// TIA Portal V20 export
TYPE "LBP_typeModularMcpUniversalInput"
TITLE = Modular MCP image / Image MCP modulaire
// Input image of universal keypad for modular MCP / Image des entrées du pupitre universel pour MCP modulaires
   STRUCT
      key0 : Bool;   // input image n+0 bit 0 / Image des entrées n+0 bit 0
      key1 : Bool;   // input image n+0 bit 1 / Image des entrées n+0 bit 1
      key2 : Bool;   // input image n+0 bit 2 / Image des entrées n+0 bit 2
      key3 : Bool;   // input image n+0 bit 3 / Image des entrées n+0 bit 3
      key4 : Bool;   // input image n+0 bit 4 / Image des entrées n+0 bit 4
      key5 : Bool;   // input image n+0 bit 5 / Image des entrées n+0 bit 5
      key6 : Bool;   // input image n+0 bit 6 / Image des entrées n+0 bit 6
      key7 : Bool;   // input image n+0 bit 7 / Image des entrées n+0 bit 7
      key8 : Bool;   // input image n+1 bit 0 / Image des entrées n+1 bit 0
      key9 : Bool;   // input image n+1 bit 1 / Image des entrées n+1 bit 1
      key10 : Bool;   // input image n+1 bit 2 / Image des entrées n+1 bit 2
      key11 : Bool;   // input image n+1 bit 3 / Image des entrées n+1 bit 3
      key12 : Bool;   // input image n+1 bit 4 / Image des entrées n+1 bit 4
      key13 : Bool;   // input image n+1 bit 5 / Image des entrées n+1 bit 5
      key14 : Bool;   // input image n+1 bit 6 / Image des entrées n+1 bit 6
      reserved17 : Bool;
      key16 : Bool;   // input image n+2 bit 0 / Image des entrées n+2 bit 0
      key17 : Bool;   // input image n+2 bit 1 / Image des entrées n+2 bit 1
      key18 : Bool;   // input image n+2 bit 2 / Image des entrées n+2 bit 2
      reserved23 : Bool;
      reserved24 : Bool;
      reserved25 : Bool;
      reserved26 : Bool;
      reserved27 : Bool;
      key24 : Bool;   // input image n+3 bit 0 / Image des entrées n+3 bit 0
      key25 : Bool;   // input image n+3 bit 1 / Image des entrées n+3 bit 1
      key26 : Bool;   // input image n+3 bit 2 / Image des entrées n+3 bit 2
      reserved33 : Bool;
      reserved34 : Bool;
      reserved35 : Bool;
      reserved36 : Bool;
      reserved37 : Bool;
   END_STRUCT;
END_TYPE
